{attribute 'GeneratedUsingTerminal: EK1100-0000-0018'}
{attribute addProperty BoxType "EK1100-0000-0018"}
{attribute addProperty Id "Beckhoff_EL3xxxEK1122Beckhoff_EL3xxxEK1122_31431A032A_0001_EL3602_0000_0016EL3602_3048840034A_0002_EL3602_0000_0017EL3602_3048840034A_0003_EL3602_0000_0018EL3602_3048840034A_0004_EL3602_0000_0019EL3602_3048840034A_0005_EL3602_0002_0016EL3602_244E2D8634A_0006_EL3602_0002_0017EL3602_244E2D8634A_0007_EL3602_0002_0018EL3602_244E2D8634A_0008_EL3602_0010_0016EL3602_3048840034A_0009_EL3602_0010_0017EL3602_3048840034A_0010_EL3602_0010_0018EL3602_3048840034A_0011_EL3602_0010_0019EL3602_3048840034A_0012_EL3602_0020_0018EL3602_244E2D8634A_0013_EL3611_1030_0016EL3611_1B2C2E2B23A_0014_EL3611_1030_0017EL3611_1B2C2E2B23A_0015_EL3612_0000_0016EL3612_3048840034A_0016_EL3612_0000_0017EL3612_3048840034A_0017_EL3612_0000_0018EL3612_3048840034A_0018_EL3612_0000_0019EL3612_3048840034A_0019_EL3612_0020_0018EL3612_3048840034A_0020_EL3612_0020_0019EL3612_3048840034A_0021_EL3621_0020_0016EL3621_1B2C2E2B23A_0022_EL3621_0020_0017EL3621_1B2C2E2B23A_0023_EL3632_0000_0016EL3632_82B2AA7686A_0024_EL3632_0000_0017EL3632_82B2AA7686A_0025_EL3632_0000_0018EL3632_82B2AA7686A_0026_EL3632_0000_0019EL3632_82B2AA7686A_0027_EL3632_0000_0020EL3632_82B2AA7686A_0028_EL3632_0000_0021EL3632_82B2AA7686A_0029_EL3632_0000_0022EL3632_A04CBB5A86A_0030_EL3632_0000_0023EL3632_A04CBB5A86A_0031_EL3681_0000_0017EL3681_9897CEC831A_0032_EL3681_0000_0018EL3681_9AA3368032A_0033_EL3681_0000_0019EL3681_9AA3368032A_0034_EL3681_0000_0020EL3681_9AA3368032A_0035_EL3681_0000_0021EL3681_B184412232A_0036_EL3692_0000_0017EL3692_CD4ED2F352A_0037_EL3692_0000_0018EL3692_CD4ED2F352A_0038_EL3692_0000_0019EL3692_CD4ED2F352A_0039_EL3692_0000_0020EL3692_CD4ED2F352A_0040_EL3692_0000_0021EL3692_CD4ED2F352"}
{attribute addProperty CRC "670531355"}
{attribute addProperty Size "1813"}
TYPE Beckhoff_EL3xxx_27F77F1B EXTENDS EK1100_AB5A9467 :
STRUCT
	{attribute addProperty Name "Beckhoff_EL3xxxEK1122"}
	{attribute addProperty PreviousPort "Beckhoff EL3xxx : B"}
	Beckhoff_EL3xxxEK1122 : Beckhoff_EL3xxxEK1122_31431A03;
	{attribute addProperty Name "A_0001_EL3602_0000_0016"}
	{attribute addProperty PreviousPort "Beckhoff EL3xxxEK1122 : C"}
	A_0001_EL3602_0000_0016 : EL3602_30488400;
	{attribute addProperty Name "A_0002_EL3602_0000_0017"}
	{attribute addProperty PreviousPort "A_0001(EL3602-0000-0016) : B"}
	A_0002_EL3602_0000_0017 : EL3602_30488400;
	{attribute addProperty Name "A_0003_EL3602_0000_0018"}
	{attribute addProperty PreviousPort "A_0002(EL3602-0000-0017) : B"}
	A_0003_EL3602_0000_0018 : EL3602_30488400;
	{attribute addProperty Name "A_0004_EL3602_0000_0019"}
	{attribute addProperty PreviousPort "A_0003(EL3602-0000-0018) : B"}
	A_0004_EL3602_0000_0019 : EL3602_30488400;
	{attribute addProperty Name "A_0005_EL3602_0002_0016"}
	{attribute addProperty PreviousPort "A_0004(EL3602-0000-0019) : B"}
	A_0005_EL3602_0002_0016 : EL3602_244E2D86;
	{attribute addProperty Name "A_0006_EL3602_0002_0017"}
	{attribute addProperty PreviousPort "A_0005(EL3602-0002-0016) : B"}
	A_0006_EL3602_0002_0017 : EL3602_244E2D86;
	{attribute addProperty Name "A_0007_EL3602_0002_0018"}
	{attribute addProperty PreviousPort "A_0006(EL3602-0002-0017) : B"}
	A_0007_EL3602_0002_0018 : EL3602_244E2D86;
	{attribute addProperty Name "A_0008_EL3602_0010_0016"}
	{attribute addProperty PreviousPort "A_0007(EL3602-0002-0018) : B"}
	A_0008_EL3602_0010_0016 : EL3602_30488400;
	{attribute addProperty Name "A_0009_EL3602_0010_0017"}
	{attribute addProperty PreviousPort "A_0008(EL3602-0010-0016) : B"}
	A_0009_EL3602_0010_0017 : EL3602_30488400;
	{attribute addProperty Name "A_0010_EL3602_0010_0018"}
	{attribute addProperty PreviousPort "A_0009(EL3602-0010-0017) : B"}
	A_0010_EL3602_0010_0018 : EL3602_30488400;
	{attribute addProperty Name "A_0011_EL3602_0010_0019"}
	{attribute addProperty PreviousPort "A_0010(EL3602-0010-0018) : B"}
	A_0011_EL3602_0010_0019 : EL3602_30488400;
	{attribute addProperty Name "A_0012_EL3602_0020_0018"}
	{attribute addProperty PreviousPort "A_0011(EL3602-0010-0019) : B"}
	A_0012_EL3602_0020_0018 : EL3602_244E2D86;
	{attribute addProperty Name "A_0013_EL3611_1030_0016"}
	{attribute addProperty PreviousPort "A_0012(EL3602-0020-0018) : B"}
	A_0013_EL3611_1030_0016 : EL3611_1B2C2E2B;
	{attribute addProperty Name "A_0014_EL3611_1030_0017"}
	{attribute addProperty PreviousPort "A_0013(EL3611-1030-0016) : B"}
	A_0014_EL3611_1030_0017 : EL3611_1B2C2E2B;
	{attribute addProperty Name "A_0015_EL3612_0000_0016"}
	{attribute addProperty PreviousPort "A_0014(EL3611-1030-0017) : B"}
	A_0015_EL3612_0000_0016 : EL3612_30488400;
	{attribute addProperty Name "A_0016_EL3612_0000_0017"}
	{attribute addProperty PreviousPort "A_0015(EL3612-0000-0016) : B"}
	A_0016_EL3612_0000_0017 : EL3612_30488400;
	{attribute addProperty Name "A_0017_EL3612_0000_0018"}
	{attribute addProperty PreviousPort "A_0016(EL3612-0000-0017) : B"}
	A_0017_EL3612_0000_0018 : EL3612_30488400;
	{attribute addProperty Name "A_0018_EL3612_0000_0019"}
	{attribute addProperty PreviousPort "A_0017(EL3612-0000-0018) : B"}
	A_0018_EL3612_0000_0019 : EL3612_30488400;
	{attribute addProperty Name "A_0019_EL3612_0020_0018"}
	{attribute addProperty PreviousPort "A_0018(EL3612-0000-0019) : B"}
	A_0019_EL3612_0020_0018 : EL3612_30488400;
	{attribute addProperty Name "A_0020_EL3612_0020_0019"}
	{attribute addProperty PreviousPort "A_0019(EL3612-0020-0018) : B"}
	A_0020_EL3612_0020_0019 : EL3612_30488400;
	{attribute addProperty Name "A_0021_EL3621_0020_0016"}
	{attribute addProperty PreviousPort "A_0020(EL3612-0020-0019) : B"}
	A_0021_EL3621_0020_0016 : EL3621_1B2C2E2B;
	{attribute addProperty Name "A_0022_EL3621_0020_0017"}
	{attribute addProperty PreviousPort "A_0021(EL3621-0020-0016) : B"}
	A_0022_EL3621_0020_0017 : EL3621_1B2C2E2B;
	{attribute addProperty Name "A_0023_EL3632_0000_0016"}
	{attribute addProperty PreviousPort "A_0022(EL3621-0020-0017) : B"}
	A_0023_EL3632_0000_0016 : EL3632_82B2AA76;
	{attribute addProperty Name "A_0024_EL3632_0000_0017"}
	{attribute addProperty PreviousPort "A_0023(EL3632-0000-0016) : B"}
	A_0024_EL3632_0000_0017 : EL3632_82B2AA76;
	{attribute addProperty Name "A_0025_EL3632_0000_0018"}
	{attribute addProperty PreviousPort "A_0024(EL3632-0000-0017) : B"}
	A_0025_EL3632_0000_0018 : EL3632_82B2AA76;
	{attribute addProperty Name "A_0026_EL3632_0000_0019"}
	{attribute addProperty PreviousPort "A_0025(EL3632-0000-0018) : B"}
	A_0026_EL3632_0000_0019 : EL3632_82B2AA76;
	{attribute addProperty Name "A_0027_EL3632_0000_0020"}
	{attribute addProperty PreviousPort "A_0026(EL3632-0000-0019) : B"}
	A_0027_EL3632_0000_0020 : EL3632_82B2AA76;
	{attribute addProperty Name "A_0028_EL3632_0000_0021"}
	{attribute addProperty PreviousPort "A_0027(EL3632-0000-0020) : B"}
	A_0028_EL3632_0000_0021 : EL3632_82B2AA76;
	{attribute addProperty Name "A_0029_EL3632_0000_0022"}
	{attribute addProperty PreviousPort "A_0028(EL3632-0000-0021) : B"}
	A_0029_EL3632_0000_0022 : EL3632_A04CBB5A;
	{attribute addProperty Name "A_0030_EL3632_0000_0023"}
	{attribute addProperty PreviousPort "A_0029(EL3632-0000-0022) : B"}
	A_0030_EL3632_0000_0023 : EL3632_A04CBB5A;
	{attribute addProperty Name "A_0031_EL3681_0000_0017"}
	{attribute addProperty PreviousPort "A_0030(EL3632-0000-0023) : B"}
	A_0031_EL3681_0000_0017 : EL3681_9897CEC8;
	{attribute addProperty Name "A_0032_EL3681_0000_0018"}
	{attribute addProperty PreviousPort "A_0031(EL3681-0000-0017) : B"}
	A_0032_EL3681_0000_0018 : EL3681_9AA33680;
	{attribute addProperty Name "A_0033_EL3681_0000_0019"}
	{attribute addProperty PreviousPort "A_0032(EL3681-0000-0018) : B"}
	A_0033_EL3681_0000_0019 : EL3681_9AA33680;
	{attribute addProperty Name "A_0034_EL3681_0000_0020"}
	{attribute addProperty PreviousPort "A_0033(EL3681-0000-0019) : B"}
	A_0034_EL3681_0000_0020 : EL3681_9AA33680;
	{attribute addProperty Name "A_0035_EL3681_0000_0021"}
	{attribute addProperty PreviousPort "A_0034(EL3681-0000-0020) : B"}
	A_0035_EL3681_0000_0021 : EL3681_B1844122;
	{attribute addProperty Name "A_0036_EL3692_0000_0017"}
	{attribute addProperty PreviousPort "A_0035(EL3681-0000-0021) : B"}
	A_0036_EL3692_0000_0017 : EL3692_CD4ED2F3;
	{attribute addProperty Name "A_0037_EL3692_0000_0018"}
	{attribute addProperty PreviousPort "A_0036(EL3692-0000-0017) : B"}
	A_0037_EL3692_0000_0018 : EL3692_CD4ED2F3;
	{attribute addProperty Name "A_0038_EL3692_0000_0019"}
	{attribute addProperty PreviousPort "A_0037(EL3692-0000-0018) : B"}
	A_0038_EL3692_0000_0019 : EL3692_CD4ED2F3;
	{attribute addProperty Name "A_0039_EL3692_0000_0020"}
	{attribute addProperty PreviousPort "A_0038(EL3692-0000-0019) : B"}
	A_0039_EL3692_0000_0020 : EL3692_CD4ED2F3;
	{attribute addProperty Name "A_0040_EL3692_0000_0021"}
	{attribute addProperty PreviousPort "A_0039(EL3692-0000-0020) : B"}
	A_0040_EL3692_0000_0021 : EL3692_CD4ED2F3;
END_STRUCT
END_TYPE

(* stored: Version 1.2.0.0, ProductVersion 3.1.4024.9
   DUT Beckhoff_EL3xxx_27F77F1B: Id {41f68ce7-720a-4fc8-88f0-e9413f01ce78} *)
